// TIA Portal V16 export
// export: Created 2024-12-03T15:41:45.2187987Z, ExportSetting WithReadOnly, DisplayName Totally Integrated Automation Portal, DisplayVersion V16 Update 6, DisplayName TIA Portal Version Control Interface, DisplayVersion V16 Update 2, DisplayName TIA Portal Openness, DisplayVersion V16 Update 6, DisplayName TIA Portal Teamcenter Gateway, DisplayVersion V16, DisplayName SINAMICS Startdrive Advanced, DisplayVersion V16 Update 5, DisplayName SINAMICS Startdrive G130, G150, S120, S150, SINAMICS MV, S210, DisplayVersion V16 Update 5, DisplayName SINAMICS Startdrive G110M, G120, G120C, G120D, G120P, G115D, DisplayVersion V16 Update 5, DisplayName STEP 7 Professional, DisplayVersion V16 Update 6, DisplayName STEP 7 Safety, DisplayVersion V16, DisplayName WinCC Advanced / Unified PC, DisplayVersion V16 Update 6
TYPE "SAI_MB_DeviceStatus"
// stored: CreationDate 2022-02-16T11:31:07.6486039Z, InterfaceModifiedDate 2020-03-20T04:25:57.9747125Z, IsConsistent true, LibraryConformanceStatus The object is library-conformant., ModifiedDate 2020-03-20T04:25:57.9747125Z
   STRUCT
      "Alternate weight unit" : Bool;
      "Run flat" : Bool;
      "Device specific bit 2" : Bool;
      "Device specific bit 3" : Bool;
      "Device specific bit 4" : Bool;
      "Device specific bit 5" : Bool;
      "Device specific bit 6" : Bool;
      "Device specific bit 7" : Bool;
      "Sequence bit 0" : Bool;
      "Sequence bit 1" : Bool;
      "Heart Beat" : Bool;
      "Data OK" : Bool;
      "Alarm Condition" : Bool;
      "Center of Zero" : Bool;
      Motion : Bool;
      "Net Mode" : Bool;
   END_STRUCT;
END_TYPE
